(* IEC 61131-3 sources: POMIRTS_lab3/AS/Library/AsMath, 2 files *)

(* ---- AsMath.fun ---- *)
(********************************************************************
 * COPYRIGHT -- Bernecker + Rainer
 ********************************************************************
 * Library: AsMath
 * File: AsMath.fun
 * Author: B+R
 ********************************************************************
 * Functions and function blocks of library AsMath
 ********************************************************************)

FUNCTION atan2 : REAL                  (*calculates the arc tangent of y/x*)
	VAR_INPUT
		y	:REAL;                     (*y*)
		x	:REAL;                     (*x*)
	END_VAR
END_FUNCTION

FUNCTION ceil : REAL                   (*calculates the smallest integer value which is greater than or equal to the input value*)
	VAR_INPUT
		x	:REAL;                     (*input value*)
	END_VAR
END_FUNCTION

FUNCTION cosh : REAL                   (*calculates the hyperbolic cosine of x*)
	VAR_INPUT
		x	:REAL;                     (*input value*)
	END_VAR
END_FUNCTION

FUNCTION floor : REAL                  (*calculates the largest integer value which is less than or equal to the input value*)
	VAR_INPUT
		x	:REAL;                     (*input value*)
	END_VAR
END_FUNCTION

FUNCTION fmod : REAL                   (*calculates the remainder of the division x/y*)
	VAR_INPUT
		x	:REAL;                     (*numerator*)
		y	:REAL;                     (*denominator*)
	END_VAR
END_FUNCTION

FUNCTION frexp : REAL                  (*calculates the mantissa and the exponent of a floating point number*)
	VAR_INPUT
		x	:REAL;                     (*input value*)
		pExp	:UDINT;                (*address of the exponent (address of DINT) (base 2)*)
	END_VAR
END_FUNCTION

FUNCTION ldexp : REAL                  (*calculates a floating point number from mantissa x and exponent exp*)
	VAR_INPUT
		x	:REAL;                     (*mantissa*)
		exp_val	:DINT;                 (*exponent (base 2)*)
	END_VAR
END_FUNCTION

FUNCTION modf : REAL                   (*separates a floating point number into an integer and decimal part*)
	VAR_INPUT
		x	:REAL;                     (*input value*)
		plp	:UDINT;                    (*address of the integer part (address of a REAL value)*)
	END_VAR
END_FUNCTION

FUNCTION pow : REAL                    (*calculates x raised to the power of y*)
	VAR_INPUT
		x	:REAL;                     (*base*)
		y	:REAL;                     (*exponent*)
	END_VAR
END_FUNCTION

FUNCTION sinh : REAL                   (*calculates the hyperbolic sine of x*)
	VAR_INPUT
		x	:REAL;                     (*input value*)
	END_VAR
END_FUNCTION

FUNCTION tanh : REAL                   (*calculates the hyperbolic tangent of x*)
	VAR_INPUT
		x	:REAL;                     (*input value*)
	END_VAR
END_FUNCTION

(* ---- AsMath.var ---- *)
(********************************************************************
 * COPYRIGHT -- Bernecker + Rainer
 ********************************************************************
 * Library: AsMath
 * File: AsMath.var
 * Author: B+R
 ********************************************************************
 * Local variables of library AsMath
 ********************************************************************)

VAR CONSTANT
	am2_SQRTPI	: REAL	:= 1.12838;    (*2/(square root from PI)*)
	amSQRT1_2	: REAL	:= 0.707107;   (*square root from 1/2*)
	amSQRTPI	: REAL	:= 1.77245;    (*square root from PI*)
	amLOG2_E	: REAL	:= 0.693147;   (*log with the base 2 from E*)
	amLOG10E	: REAL	:= 0.434294;   (*log with the base 10 from E*)
	amIVLN10	: REAL	:= 0.434294;   (*1/(ln from 10)*)
	amINVLN2	: REAL	:=  1.4427;    (*1/(ln from 2)*)
	amTWOPI	: REAL	:= 6.28319;        (*2 PI*)
	amSQRT3	: REAL	:= 1.73205;        (*square root from 3*)
	amSQRT2	: REAL	:= 1.41421;        (*square root from 2*)
	amLOG2E	: REAL	:=  1.4427;        (*log with the base 2 from E*)
	amLN2LO	: REAL	:= 1.90821e-010;   (*log with the base 2 from LOW*)
	amLN2HI	: REAL	:= 0.693147;       (*log with the base 2 from HIGH*)
	am3PI_4	: REAL	:= 2.35619;        (*3/4 PI*)
	amPI_4	: REAL	:= 0.785398;       (*PI/4*)
	amPI_2	: REAL	:=  1.5708;        (*PI/2*)
	amLN10	: REAL	:= 2.30259;        (*ln from 10*)
	am2_PI	: REAL	:= 0.63662;        (*2/PI*)
	am1_PI	: REAL	:= 0.31831;        (*1/PI*)
	amLN2	: REAL	:= 0.693147;       (*ln from 2*)
	amPI	: REAL	:= 3.14159;        (*PI*)
	amE	: REAL	:= 2.71828;            (*E*)
END_VAR
